(*
Specifies the anti-windup behaviour of :class:`FB_ClampingIntegrator` when
saturation is detected via :attr:`~FB_ClampingIntegrator.ComparitorInput`.
*)
{attribute 'qualified_only'}
{attribute 'strict'}
{attribute 'to_string'}
TYPE E_AntiWindupMode :
(
	// Holds the integrator output at its current value while saturation is active.
	Hold := 0,
	// Zeroes the integrator output on the rising edge of saturation detection.
	Off  := 1
)BYTE;
END_TYPE

(* stored: Version 1.1.0.1, ProductVersion 3.1.4024.15
   EnumerationTextList E_AntiWindupMode: Id {d454041f-725a-4fd9-8138-fb1750f0ea89} *)
